# EPICS substitutions: testioApp/Db/input.substitutions
file ../../db/input.db {
    pattern	{Sys,	  	Pin, 	Scan,		Desc}
		{"BBB01",	"1",	"1 second"	"Adc 1 BeagleBone"}
}
